# EPICS autosave request: as/req/modules_ANC300.req
#FILE... modules_ANC300.req

file "ANC300.req", DEVICE=E1:ANC300
